// TIA Portal V19 export
TYPE "LEXCHANGETRAY_typeRollerIoSignalConfigeration_B2"
// referenceDesignator: String[20]
// simActive: Bool
// stored: Access Published
   STRUCT
      referenceDesignator : String[20] := 'U3Em1IO';
      simActive : Bool;
   END_STRUCT;
END_TYPE
